FUNCTION CheckDivDint : DINT
VAR_INPUT
	divisor				: DINT;
END_VAR
VAR
END_VAR

IF divisor = 0 THEN
	CheckDintZeroDiv_ErrCnt:= CheckDintZeroDiv_ErrCnt + 1;
	CheckDivDint := 1;
ELSE
	CheckDivDint := divisor;
END_IF

END_FUNCTION

(* stored: Version 1.1.0.1, ProductVersion 3.1.4024.9
   POU CheckDivDint: Id {74cf1fae-c527-4cba-83bf-86a6548a15dd}, SpecialFunc CheckDivInt32 *)
